// TwinCAT 3 PLC project FMEvents
// Title: FM Events
// Company: FrameworkMonorepo
// ProjectVersion: 0.0.1
// ProgramVersion: 3.1.4024.0
// libraries:
//   FM Common Interfaces, * (FrameworkMonorepo)
//   Tc3_EventLogger, * (Beckhoff Automation GmbH)
// project tree:
//   EventManager/ EventLoggerManager.TcPOU, EventManager.TcIO
//   / EventParameters.TcGVL
//   Event/ AlarmEventLogger.TcPOU, Alarm.TcIO, Message.TcIO, MessageEventLogger.TcPOU
//   Version/ Global_Version.TcGVL
// (motion and I/O tree: see PLC project fmtypes)
// real-time tasks:
//   TASK BindingTestTask: cycle T#1ms, priority 20, ADS port 350
//   TASK PlcTask: cycle T#1ms, priority 21, ADS port 351
//   TASK PlcTask1: cycle T#1ms, priority 22, ADS port 352
//   TASK PlcTask2: cycle T#1ms, priority 23, ADS port 353
//   TASK MathTestTask: cycle T#1ms, priority 24, ADS port 354
//   TASK TimesTestsTask: cycle T#1ms, priority 25, ADS port 355

// ---- EventParameters.TcGVL
{attribute 'qualified_only'}
VAR_GLOBAL CONSTANT
	EscapeBackslash : BOOL := FALSE;
END_VAR

// ---- Version/Global_Version.TcGVL
{attribute 'TcGenerated'}
{attribute 'no-analysis'}
{attribute 'linkalways'}
// This function has been automatically generated from the project information.
VAR_GLOBAL CONSTANT
	{attribute 'const_non_replaced'}
	stLibVersion_FM_Events : ST_LibVersion := (iMajor := 0, iMinor := 0, iBuild := 1, iRevision := 0, nFlags := 0, sVersion := '0.0.1');
END_VAR

// ---- EventManager/EventManager.TcIO
INTERFACE EventManager

METHOD ClearAll
VAR_INPUT
END_VAR
END_METHOD

END_INTERFACE

// ---- Event/Alarm.TcIO
INTERFACE Alarm

METHOD Clear
VAR_INPUT
END_VAR
END_METHOD

METHOD ClearArguments : I_TcArguments
END_METHOD

{attribute 'monitoring' := 'call'}
PROPERTY IsRaised : BOOL
GET
END_GET
END_PROPERTY

METHOD Raise
VAR_INPUT
END_VAR
END_METHOD

{attribute 'monitoring' := 'call'}
PROPERTY Source : Name
GET
END_GET
SET
END_SET
END_PROPERTY

END_INTERFACE

// ---- Event/Message.TcIO
INTERFACE Message

METHOD ClearArguments : I_TcArguments
END_METHOD

METHOD Send
VAR_INPUT
END_VAR
END_METHOD

{attribute 'monitoring' := 'call'}
PROPERTY Source : Name
GET
END_GET
SET
END_SET
END_PROPERTY

END_INTERFACE

// ---- EventManager/EventLoggerManager.TcPOU
FUNCTION_BLOCK EventLoggerManager IMPLEMENTS EventManager
VAR
	eventLogger : FB_TcEventLogger;
END_VAR

METHOD ClearAll
VAR_INPUT
END_VAR
eventLogger.ClearAlarms(0, TRUE, 0);
END_METHOD

END_FUNCTION_BLOCK

// ---- Event/AlarmEventLogger.TcPOU
FUNCTION_BLOCK AlarmEventLogger IMPLEMENTS Alarm
VAR
	alarm : FB_TcAlarm;
	_Source : Name;
	autoReset : BOOL;
END_VAR

PROPERTY Arguments : I_TcArguments
GET
Arguments := alarm.ipArguments;
END_GET
END_PROPERTY

METHOD Clear
VAR_INPUT
END_VAR
alarm.Clear(0, TRUE);
END_METHOD

METHOD ClearArguments : I_TcArguments
alarm.ipArguments.Clear();

IF (_Source <> 0) THEN
	alarm.ipArguments.AddStringByValue(value := _Source.Name);
END_IF

ClearArguments := alarm.ipArguments;
END_METHOD

METHOD FB_init : BOOL
VAR_INPUT
	bInitRetains : BOOL; // if TRUE, the retain variables are initialized (warm start / cold start)
	bInCopyCode : BOOL;  // if TRUE, the instance afterwards gets moved into the copy code (online change)
	
	event : TcEventEntry;
	autoReset : BOOL;
END_VAR
THIS^.autoReset := autoReset;
alarm.CreateEx(stEventEntry := event, bWithConfirmation := NOT autoReset, ipSourceInfo := 0);
END_METHOD

{attribute 'monitoring' := 'call'}
PROPERTY IsRaised : BOOL
GET
IsRaised := alarm.bRaised;
END_GET
END_PROPERTY

METHOD Raise
VAR_INPUT
END_VAR
IF (alarm.ipArguments.nCount = 0 AND _Source <> 0) THEN
	alarm.ipArguments.AddStringByValue(value := _Source.Name);
END_IF

alarm.Raise(0);
END_METHOD

{attribute 'monitoring' := 'call'}
PROPERTY Source : Name
GET
Source := _Source;
END_GET
SET
_Source := Source;
END_SET
END_PROPERTY

METHOD Watch
VAR_INPUT
	eventCondition : BOOL;
END_VAR
IF (eventCondition) THEN
	Raise();
ELSIF (autoReset AND IsRaised) THEN
	Clear();
END_IF
END_METHOD

END_FUNCTION_BLOCK

// ---- Event/MessageEventLogger.TcPOU
FUNCTION_BLOCK MessageEventLogger IMPLEMENTS Message
VAR
	message : FB_TcMessage;
	_Source : Name;
END_VAR

PROPERTY Arguments : I_TcArguments
GET
Arguments := message.ipArguments;
END_GET
END_PROPERTY

METHOD ClearArguments : I_TcArguments
message.ipArguments.Clear();

IF (_Source <> 0) THEN
	message.ipArguments.AddStringByValue(value := _Source.Name);
END_IF

ClearArguments := message.ipArguments;
END_METHOD

METHOD FB_init : BOOL
VAR_INPUT
	bInitRetains : BOOL; // if TRUE, the retain variables are initialized (warm start / cold start)
	bInCopyCode : BOOL;  // if TRUE, the instance afterwards gets moved into the copy code (online change)
	
	event : TcEventEntry;
END_VAR
message.CreateEx(stEventEntry := event, ipSourceInfo := 0);
END_METHOD

METHOD Send
VAR_INPUT
END_VAR
IF (message.ipArguments.nCount = 0 AND _Source <> 0) THEN
	message.ipArguments.AddStringByValue(value := _Source.Name);
END_IF

message.Send(0);
END_METHOD

{attribute 'monitoring' := 'call'}
PROPERTY Source : Name
GET
Source := _Source;
END_GET
SET
_Source := Source;
END_SET
END_PROPERTY

METHOD Watch
VAR_INPUT
	eventCondition : BOOL;
END_VAR
IF (eventCondition) THEN
	Send();
END_IF
END_METHOD

END_FUNCTION_BLOCK
